// TIA Portal V21 export
DATA_BLOCK "HmiTags"   // DB16
{ S7_Optimized_Access := 'FALSE' }
// stored: AutoNumber false
   VAR
      MasterReset : Bool;
      SystemRestart : Bool;
      ManualModeFAULT : Bool;
      AlarmAck : Bool;
      Hooter : Bool;
      ResetButton : Bool;
      VesselStatus : Int;
      Weight_int : Int;
      Weight_Temp : Real;
      VesselMaxPressure : Real := 5.0;
      CycleDataLog : Bool;
      CyclePrintData : Bool;
      AlarmPath : String := '/media/simatic/data-storage/Reports/Pdf/Alarm.pdf';
      HelpPath : String := ' /media/simatic/data-storage/OPM/R-OPM.pdf';
      AlarmStarTime : DTL;
      AlarmEndTime : DTL;
      EpoxyMMActual { S7_SetPoint := 'True'} : Real;
      PlcHmiComBreak : Bool;
      AuditStartTime : DTL;
      AuditEndTime : DTL;
      AuditPath : String := '/media/simatic/data-storage/Reports/Pdf/Audit.pdf';
      UserAuditStartTime : DTL;
      UserAuditEndTime : DTL;
      UserAuditPath : String := '/media/simatic/data-storage/Reports/Pdf/UserAudit.pdf';
      LF_time_delay : Int;
      JacketRecoveryCycSelected : Bool;
      JacketRecoveryFault : Bool;
      JacketRecoveryCycEnable : Bool;
      pulse : Array[0..14] of Bool;
      BatchDetailsBlankPopup : Bool;
      BatchDetailsBlankPopupAck : Bool;
      AccessTablePath : String := '/media/simatic/data-storage/Reports/Pdf/AccessTable.pdf';
      LoadCellResult : String;
   END_VAR
BEGIN
END_DATA_BLOCK
